Staubli VAL3: CompareTwoJoint.pgx

public program CompareTwoJoint(joint x_jFirst, joint x_jSecond, bool& x_bSame, bool x_bIs6Axis)
  local joint l_jTolerance
begin
  //比较两个关节点是否相等
  x_bSame=false
  if x_bIs6Axis
    //六轴
    l_jTolerance={0.1,0.1,0.1,0.1}
    if abs(x_jFirst-x_jSecond)<l_jTolerance
        x_bSame=true
        return
    endIf
  else
    //四轴
    l_jTolerance={0.1,0.1,0.1,0.1,0.1,0.1}
    if abs(x_jFirst-x_jSecond)<l_jTolerance
        x_bSame=true
        return
    endIf
  endIf
end
